// TIA Portal V17 program export: 1 tag tables, 0 data types, 3 data blocks, 7 code blocks (in call order from the OBs), 5 instance data blocks

VAR_GLOBAL   // PLC tag table "Default tag table"
   System_Byte AT %MB1 : Byte;
   FirstScan AT %M1.0 : Bool;
   DiagStatusUpdate AT %M1.1 : Bool;
   AlwaysTRUE AT %M1.2 : Bool;
   AlwaysFALSE AT %M1.3 : Bool;
   Clock_Byte AT %MB0 : Byte;
   Clock_10Hz AT %M0.0 : Bool;
   Clock_5Hz AT %M0.1 : Bool;
   "Clock_2.5Hz" AT %M0.2 : Bool;
   Clock_2Hz AT %M0.3 : Bool;
   "Clock_1.25Hz" AT %M0.4 : Bool;
   Clock_1Hz AT %M0.5 : Bool;
   "Clock_0.625Hz" AT %M0.6 : Bool;
   "Clock_0.5Hz" AT %M0.7 : Bool;
   lastEncoderValue AT %MW8 : Int;
   encoderNumberOfTurn AT %MD10 : DInt;
   machinePosition AT %MD14 : DInt;
   goToPosition AT %M2.0 : Bool;
   broken0 AT %Q0.0 : Bool;
   broken1 AT %Q0.1 : Bool;
   baseSensor AT %I0.0 : Bool;
   stepperMotor_Direction AT %Q0.3 : Bool;
   stepperMotor_Pulse AT %Q0.2 : Bool;
   jogBackward AT %M2.1 : Bool;
   baseReq AT %M2.2 : Bool;
   jogBackwardFromSetpoint AT %M2.3 : Bool;
   jogForward AT %M2.4 : Bool;
   jogForwardFromSetpoint AT %M2.5 : Bool;
   memoryBit0 AT %M2.6 : Bool;
   memoryBit1 AT %M2.7 : Bool;
   inPosition AT %M3.0 : Bool;
   memoryBit2 AT %M3.1 : Bool;
   memoryBit3 AT %M3.2 : Bool;
   homing AT %M3.3 : Bool;
   homingDone AT %M3.4 : Bool;
   memoryBit4 AT %M3.5 : Bool;
   memoryBit5 AT %M3.6 : Bool;
   homingStep1 AT %M3.7 : Bool;
   homingStep2 AT %M4.0 : Bool;
   memoryBit6 AT %M4.1 : Bool;
   homingStep3 AT %M4.2 : Bool;
   memoryBit7 AT %M4.3 : Bool;
   seqNum AT %MW6 : Int;
   memoryBit8 AT %M4.4 : Bool;
   memoryBit9 AT %M4.5 : Bool;
   memoryBit10 AT %M4.6 : Bool;
   checkPositionAfterReboot AT %M4.7 : Bool;
   memoryBit11 AT %M5.0 : Bool;
   positionNotActual AT %M5.1 : Bool;
END_VAR

DATA_BLOCK "HMI"   // DB2
{ S7_Optimized_Access := 'FALSE' }
VERSION : 0.1
// stored: AutoNumber true, DBAccessibleFromOPCUA true, IsOnlyStoredInLoadMemory false, IsWriteProtectedInAS false
   VAR RETAIN
      sensor : Bool := 1;
      machinePosition : DInt := 77;
      encoderTurn : DInt := 20;
      encoderPosition : Int;
      setpoint : Int;
      buttonBase : Bool;
      buttonStart : Bool;
      buttonStop : Bool;
      jogBackward : Bool;
      jogForward : Bool;
      jogVelocity : Int := 50;
      machineVelocity : Int := 70;
      baseVelocity : Int := 20;
      machineConst : DInt := 42625;   // numberOfpulseEncoder 1023 numberOfTurnPer90st 2,24*90
      serwisSetpointEnable : Bool;
      serwisMachineSetpoint : DInt;
   END_VAR
BEGIN
END_DATA_BLOCK

DATA_BLOCK "machineData"   // DB1
{ S7_Optimized_Access := 'TRUE' }
VERSION : 0.1
// stored: AutoNumber true, DBAccessibleFromOPCUA true, IsOnlyStoredInLoadMemory false, IsRetainMemResEnabled false, IsWriteProtectedInAS false, MemoryReserve 100
   VAR
      encoderTurn : DInt;
      reqVelocity : Real;
      encoderValue : Int;
   END_VAR
   VAR RETAIN
      machinePosition : DInt;
   END_VAR
   VAR
      direction : Bool;
   END_VAR
   VAR RETAIN
      lastEncoderValue : DInt;
      lastMachinePosition : DInt;
   END_VAR
BEGIN
END_DATA_BLOCK

DATA_BLOCK "modbus"   // DB3
{ S7_Optimized_Access := 'FALSE'; DB_Accessible_From_OPC_UA := 'FALSE' }
VERSION : 0.1
// stored: AutoNumber true, DBAccessibleFromOPCUA false, IsOnlyStoredInLoadMemory false, IsWriteProtectedInAS false
   VAR
      rs485parity : Int := 0;
      rs485baudrate : Int := 9600;
      modbusEncoderAdd : Int := 1;
      modbusMode : Int := 0;
      modbusEncoderDataRegister : DInt := 40001;
      modbusDataLength : DInt := 1;
      encoderMaxValue : DInt := 1024;
      mbLoadError : Bool;
      mbLoadDone : Bool;
      mbLoadStatus : Word;
      mbMasterBusy : Bool;
      mbMasterDone : Bool;
      mbMasterError : Bool;
      mbMasterStatus : Word;
      modbusReqBit : Bool;
      modbusReqAgainBit : Bool;
      modbusTimer : IEC_TIMER;
      REGISTERS : Array[0..9] of Int;
      lastEncoderValue : Int;
   END_VAR
BEGIN
   modbusTimer.PT := T#2S;
END_DATA_BLOCK

ORGANIZATION_BLOCK "Main"   // OB1, LAD, ProgramCycle
TITLE = "Main Program Sweep (Cycle)"
{ S7_Optimized_Access := 'TRUE' }
VERSION : 0.1
// stored: AutoNumber true, IsIECCheckEnabled false, SetENOAutomatically false
   VAR_INPUT
      Initial_Call : Bool;   // Initial call of this OB
      Remanence : Bool;   // =True, if remanent data are available
   END_VAR
   VAR_TEMP
      turn : Int;
      machinePosition : DInt;
   END_VAR
   VAR_TEMP   // added for the SCL form of the ladder/FBD networks
      _w1 : Bool;
      _w2 : Bool;
      _w3 : Bool;
   END_VAR
BEGIN

REGION Network 1: Encoder modbus function
   // te
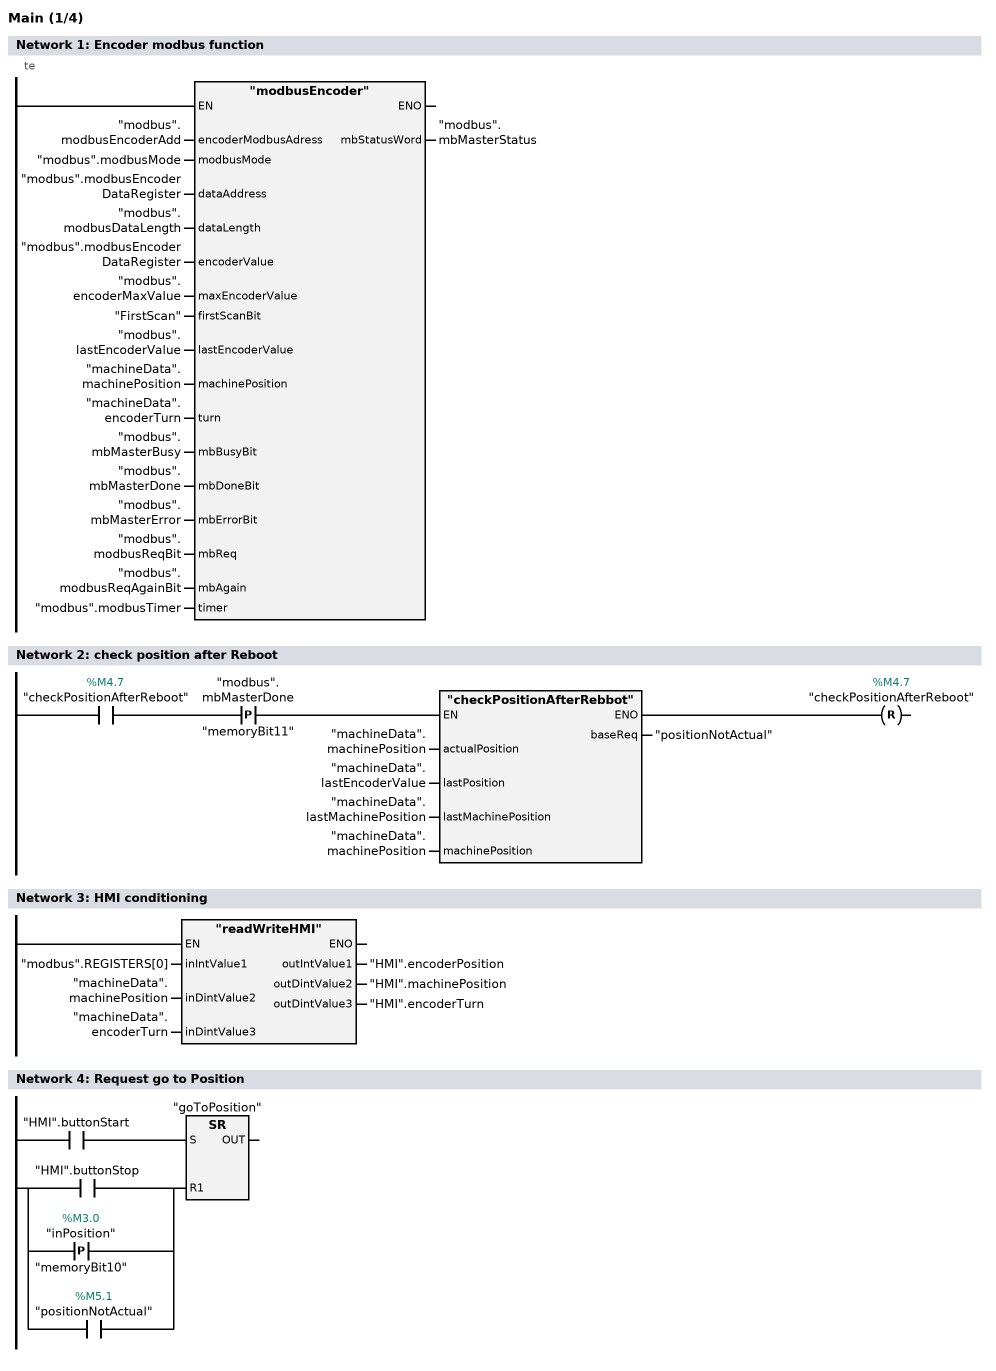
   RUNG wire#powerrail
      "modbusEncoder"(encoderModbusAdress := "modbus".modbusEncoderAdd, modbusMode := "modbus".modbusMode, dataAddress := "modbus".modbusEncoderDataRegister, dataLength := "modbus".modbusDataLength, encoderValue := "modbus".modbusEncoderDataRegister, maxEncoderValue := "modbus".encoderMaxValue, firstScanBit := "FirstScan", lastEncoderValue := "modbus".lastEncoderValue, machinePosition := "machineData".machinePosition, turn := "machineData".encoderTurn, mbBusyBit := "modbus".mbMasterBusy, mbDoneBit := "modbus".mbMasterDone, mbErrorBit := "modbus".mbMasterError, mbReq := "modbus".modbusReqBit, mbAgain := "modbus".modbusReqAgainBit, "timer" := "modbus".modbusTimer, mbStatusWord => "modbus".mbMasterStatus)
   END_RUNG
   // the same network as SCL:
   "modbusEncoder"(encoderModbusAdress := "modbus".modbusEncoderAdd,
                   modbusMode := "modbus".modbusMode,
                   dataAddress := "modbus".modbusEncoderDataRegister,
                   dataLength := "modbus".modbusDataLength,
                   encoderValue := "modbus".modbusEncoderDataRegister,
                   maxEncoderValue := "modbus".encoderMaxValue,
                   firstScanBit := "FirstScan",
                   lastEncoderValue := "modbus".lastEncoderValue,
                   machinePosition := "machineData".machinePosition,
                   turn := "machineData".encoderTurn,
                   mbBusyBit := "modbus".mbMasterBusy,
                   mbDoneBit := "modbus".mbMasterDone,
                   mbErrorBit := "modbus".mbMasterError,
                   mbReq := "modbus".modbusReqBit,
                   mbAgain := "modbus".modbusReqAgainBit,
                   "timer" := "modbus".modbusTimer,
                   mbStatusWord => "modbus".mbMasterStatus);
END_REGION

REGION Network 2: check position after Reboot
   RUNG wire#powerrail
      Contact( "checkPositionAfterReboot" )
      P_Contact(operand := "modbus".mbMasterDone, bit := "memoryBit11")
      "checkPositionAfterRebbot"(actualPosition := "machineData".machinePosition, lastPosition := "machineData".lastEncoderValue, lastMachinePosition := "machineData".lastMachinePosition, machinePosition := "machineData".machinePosition, baseReq => "positionNotActual")
      R_Coil( "checkPositionAfterReboot" )
   END_RUNG
   // the same network as SCL:
   #_w1 := "checkPositionAfterReboot" AND "modbus".mbMasterDone AND NOT "memoryBit11";   // rising edge of "modbus".mbMasterDone
   "memoryBit11" := "modbus".mbMasterDone;
   "checkPositionAfterRebbot"(EN := #_w1,
                           actualPosition := "machineData".machinePosition,
                           lastPosition := "machineData".lastEncoderValue,
                           lastMachinePosition := "machineData".lastMachinePosition,
                           machinePosition := "machineData".machinePosition,
                           baseReq => "positionNotActual",
                           ENO => #_w2);
   IF #_w2 THEN "checkPositionAfterReboot" := FALSE; END_IF;
END_REGION

REGION Network 3: HMI conditioning
   RUNG wire#powerrail
      "readWriteHMI"(inIntValue1 := "modbus".REGISTERS[0], inDintValue2 := "machineData".machinePosition, inDintValue3 := "machineData".encoderTurn, outIntValue1 => "HMI".encoderPosition, outDintValue2 => "HMI".machinePosition, outDintValue3 => "HMI".encoderTurn)
   END_RUNG
   // the same network as SCL:
   "readWriteHMI"(inIntValue1 := "modbus".REGISTERS[0],
                  inDintValue2 := "machineData".machinePosition,
                  inDintValue3 := "machineData".encoderTurn,
                  outIntValue1 => "HMI".encoderPosition,
                  outDintValue2 => "HMI".machinePosition,
                  outDintValue3 => "HMI".encoderTurn);
END_REGION

REGION Network 4: Request go to Position
   RUNG wire#powerrail
      Contact( "HMI".buttonStart )
      S_SR(operand := "goToPosition", r1 := wire#w1)
   END_RUNG
   RUNG wire#powerrail
      Contact( "HMI".buttonStop )
   END_RUNG wire#w1
   RUNG wire#powerrail
      P_Contact(operand := "inPosition", bit := "memoryBit10")
   END_RUNG wire#w1
   RUNG wire#powerrail
      Contact( "positionNotActual" )
   END_RUNG wire#w1
   // the same network as SCL:
   #_w1 := "inPosition" AND NOT "memoryBit10";   // rising edge of "inPosition"
   "memoryBit10" := "inPosition";
   IF "HMI".buttonStart THEN
       "goToPosition" := TRUE;   // SR flip-flop
   END_IF;
   IF "HMI".buttonStop OR #_w1 OR "positionNotActual" THEN "goToPosition" := FALSE; END_IF;
END_REGION

REGION Network 5: Homing
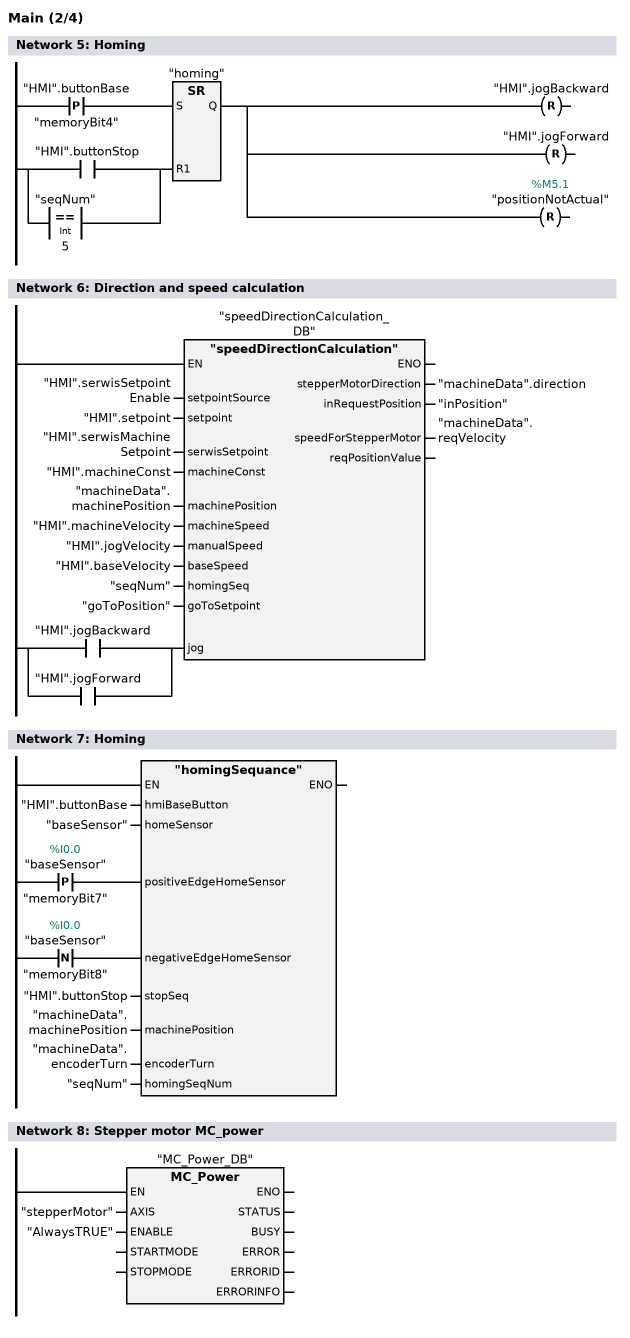
   RUNG wire#powerrail
      P_Contact(operand := "HMI".buttonBase, bit := "memoryBit4")
      S_SR(operand := "homing", r1 := wire#w1)
      wire#w2
      R_Coil( "HMI".jogBackward )
   END_RUNG
   RUNG wire#powerrail
      Contact( "HMI".buttonStop )
   END_RUNG wire#w1
   RUNG wire#powerrail
      { S7_Templates := "SrcType := Int" } EQ_Contact(in1 := "seqNum", in2 := 5)
   END_RUNG wire#w1
   RUNG wire#w2
      R_Coil( "HMI".jogForward )
   END_RUNG
   RUNG wire#w2
      R_Coil( "positionNotActual" )
   END_RUNG
   // the same network as SCL:
   #_w1 := "HMI".buttonBase AND NOT "memoryBit4";   // rising edge of "HMI".buttonBase
   "memoryBit4" := "HMI".buttonBase;
   IF #_w1 THEN
       "homing" := TRUE;   // SR flip-flop
   END_IF;
   IF "HMI".buttonStop OR ("seqNum" = 5) THEN "homing" := FALSE; END_IF;
   IF "homing" THEN
       "HMI".jogBackward := FALSE;
       "HMI".jogForward := FALSE;
       "positionNotActual" := FALSE;
   END_IF;
END_REGION

REGION Network 6: Direction and speed calculation
   RUNG wire#powerrail
      "speedDirectionCalculation_DB"(jog := wire#w1, setpointSource := "HMI".serwisSetpointEnable, setpoint := "HMI".setpoint, serwisSetpoint := "HMI".serwisMachineSetpoint, machineConst := "HMI".machineConst, machinePosition := "machineData".machinePosition, machineSpeed := "HMI".machineVelocity, manualSpeed := "HMI".jogVelocity, baseSpeed := "HMI".baseVelocity, homingSeq := "seqNum", goToSetpoint := "goToPosition", stepperMotorDirection => "machineData".direction, inRequestPosition => "inPosition", speedForStepperMotor => "machineData".reqVelocity, reqPositionValue =>)
   END_RUNG
   RUNG wire#powerrail
      Contact( "HMI".jogBackward )
   END_RUNG wire#w1
   RUNG wire#powerrail
      Contact( "HMI".jogForward )
   END_RUNG wire#w1
   // the same network as SCL:
   "speedDirectionCalculation_DB"(setpointSource := "HMI".serwisSetpointEnable,   // "speedDirectionCalculation"
                           setpoint := "HMI".setpoint,
                           serwisSetpoint := "HMI".serwisMachineSetpoint,
                           machineConst := "HMI".machineConst,
                           machinePosition := "machineData".machinePosition,
                           machineSpeed := "HMI".machineVelocity,
                           manualSpeed := "HMI".jogVelocity,
                           baseSpeed := "HMI".baseVelocity,
                           homingSeq := "seqNum",
                           goToSetpoint := "goToPosition",
                           jog := "HMI".jogBackward OR "HMI".jogForward,
                           stepperMotorDirection => "machineData".direction,
                           inRequestPosition => "inPosition",
                           speedForStepperMotor => "machineData".reqVelocity);
END_REGION

REGION Network 7: Homing
   RUNG wire#powerrail
      "homingSequance"(positiveEdgeHomeSensor := wire#w1, negativeEdgeHomeSensor := wire#w2, hmiBaseButton := "HMI".buttonBase, homeSensor := "baseSensor", stopSeq := "HMI".buttonStop, machinePosition := "machineData".machinePosition, encoderTurn := "machineData".encoderTurn, homingSeqNum := "seqNum")
   END_RUNG
   RUNG wire#powerrail
      P_Contact(operand := "baseSensor", bit := "memoryBit7")
   END_RUNG wire#w1
   RUNG wire#powerrail
      N_Contact(operand := "baseSensor", bit := "memoryBit8")
   END_RUNG wire#w2
   // the same network as SCL:
   #_w1 := "baseSensor" AND NOT "memoryBit7";   // rising edge of "baseSensor"
   "memoryBit7" := "baseSensor";
   #_w2 := NOT "baseSensor" AND "memoryBit8";   // falling edge of "baseSensor"
   "memoryBit8" := "baseSensor";
   "homingSequance"(hmiBaseButton := "HMI".buttonBase,
                    homeSensor := "baseSensor",
                    positiveEdgeHomeSensor := #_w1,
                    negativeEdgeHomeSensor := #_w2,
                    stopSeq := "HMI".buttonStop,
                    machinePosition := "machineData".machinePosition,
                    encoderTurn := "machineData".encoderTurn,
                    homingSeqNum := "seqNum");
END_REGION

REGION Network 8: Stepper motor MC_power
   RUNG wire#powerrail
      "MC_Power_DB".MC_Power(Axis := "stepperMotor", Enable := "AlwaysTRUE", StartMode :=, StopMode :=, Status =>, Busy =>, Error =>, ErrorID =>, ErrorInfo =>)
   END_RUNG
   // the same network as SCL:
   "MC_Power_DB"(Axis := "stepperMotor", Enable := "AlwaysTRUE");   // MC_Power
END_REGION

REGION Network 9: Srepper motor drive
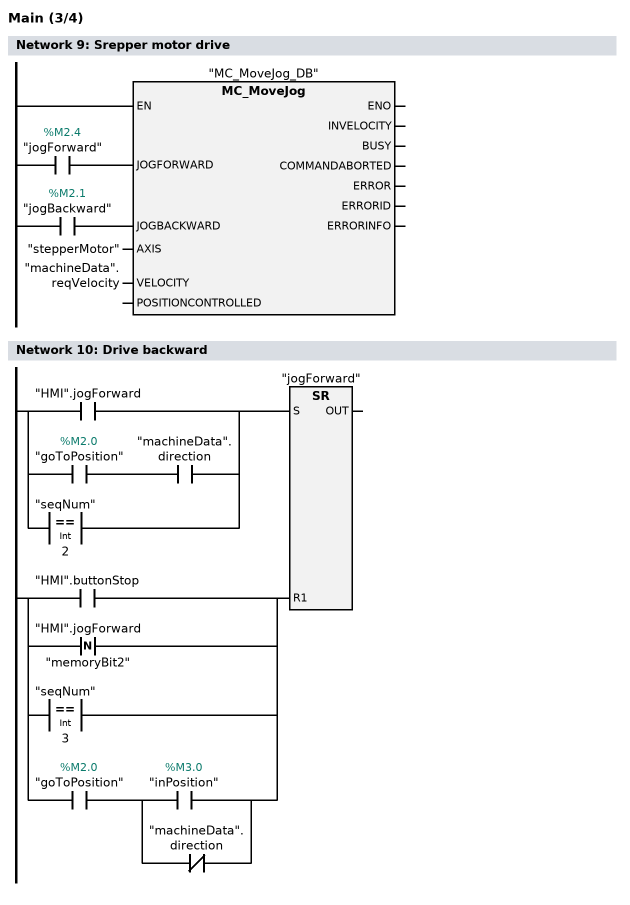
   RUNG wire#powerrail
      "MC_MoveJog_DB".MC_MoveJog(JogForward := wire#w1, JogBackward := wire#w2, Axis := "stepperMotor", Velocity := "machineData".reqVelocity, PositionControlled :=, InVelocity =>, Busy =>, CommandAborted =>, Error =>, ErrorID =>, ErrorInfo =>)
   END_RUNG
   RUNG wire#powerrail
      Contact( "jogForward" )
   END_RUNG wire#w1
   RUNG wire#powerrail
      Contact( "jogBackward" )
   END_RUNG wire#w2
   // the same network as SCL:
   "MC_MoveJog_DB"(JogForward := "jogForward",   // MC_MoveJog
                   JogBackward := "jogBackward",
                   Axis := "stepperMotor",
                   Velocity := "machineData".reqVelocity);
END_REGION

REGION Network 10: Drive backward
   RUNG wire#powerrail
      Contact( "HMI".jogForward )
      wire#w1
      S_SR(operand := "jogForward", r1 := wire#w3)
   END_RUNG
   RUNG wire#powerrail
      Contact( "goToPosition" )
      Contact( "machineData".direction )
   END_RUNG wire#w1
   RUNG wire#powerrail
      { S7_Templates := "SrcType := Int" } EQ_Contact(in1 := "seqNum", in2 := 2)
   END_RUNG wire#w1
   RUNG wire#powerrail
      Contact( "HMI".buttonStop )
   END_RUNG wire#w3
   RUNG wire#powerrail
      N_Contact(operand := "HMI".jogForward, bit := "memoryBit2")
   END_RUNG wire#w3
   RUNG wire#powerrail
      { S7_Templates := "SrcType := Int" } EQ_Contact(in1 := "seqNum", in2 := 3)
   END_RUNG wire#w3
   RUNG wire#powerrail
      Contact( "goToPosition" )
      wire#w2
      Contact( "inPosition" )
   END_RUNG wire#w3
   RUNG wire#w2
      I_Contact( "machineData".direction )
   END_RUNG wire#w3
   // the same network as SCL:
   #_w1 := NOT "HMI".jogForward AND "memoryBit2";   // falling edge of "HMI".jogForward
   "memoryBit2" := "HMI".jogForward;
   IF "HMI".jogForward OR ("goToPosition" AND "machineData".direction) OR ("seqNum" = 2) THEN
       "jogForward" := TRUE;   // SR flip-flop
   END_IF;
   IF "HMI".buttonStop OR #_w1 OR ("seqNum" = 3) OR ("goToPosition" AND ("inPosition" OR NOT "machineData".direction)) THEN
       "jogForward" := FALSE;
   END_IF;
END_REGION

REGION Network 11: Drive forward
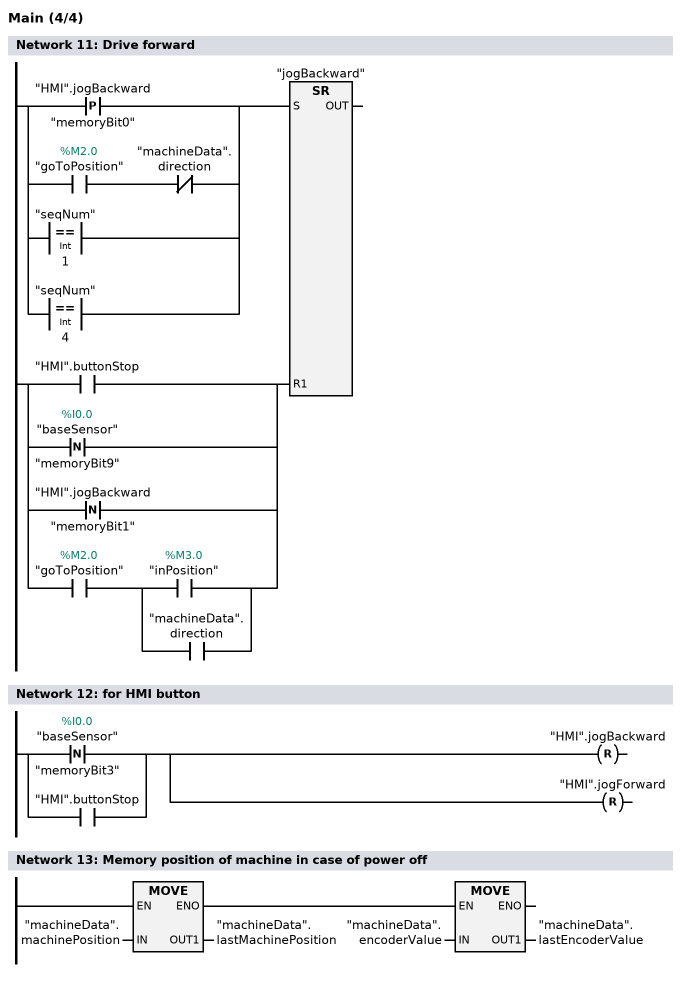
   RUNG wire#powerrail
      P_Contact(operand := "HMI".jogBackward, bit := "memoryBit0")
      wire#w1
      S_SR(operand := "jogBackward", r1 := wire#w3)
   END_RUNG
   RUNG wire#powerrail
      Contact( "goToPosition" )
      I_Contact( "machineData".direction )
   END_RUNG wire#w1
   RUNG wire#powerrail
      { S7_Templates := "SrcType := Int" } EQ_Contact(in1 := "seqNum", in2 := 1)
   END_RUNG wire#w1
   RUNG wire#powerrail
      { S7_Templates := "SrcType := Int" } EQ_Contact(in1 := "seqNum", in2 := 4)
   END_RUNG wire#w1
   RUNG wire#powerrail
      Contact( "HMI".buttonStop )
   END_RUNG wire#w3
   RUNG wire#powerrail
      N_Contact(operand := "baseSensor", bit := "memoryBit9")
   END_RUNG wire#w3
   RUNG wire#powerrail
      N_Contact(operand := "HMI".jogBackward, bit := "memoryBit1")
   END_RUNG wire#w3
   RUNG wire#powerrail
      Contact( "goToPosition" )
      wire#w2
      Contact( "inPosition" )
   END_RUNG wire#w3
   RUNG wire#w2
      Contact( "machineData".direction )
   END_RUNG wire#w3
   // the same network as SCL:
   #_w1 := "HMI".jogBackward AND NOT "memoryBit0";   // rising edge of "HMI".jogBackward
   "memoryBit0" := "HMI".jogBackward;
   #_w2 := NOT "baseSensor" AND "memoryBit9";   // falling edge of "baseSensor"
   "memoryBit9" := "baseSensor";
   #_w3 := NOT "HMI".jogBackward AND "memoryBit1";   // falling edge of "HMI".jogBackward
   "memoryBit1" := "HMI".jogBackward;
   IF #_w1 OR ("goToPosition" AND NOT "machineData".direction) OR ("seqNum" = 1) OR ("seqNum" = 4) THEN
       "jogBackward" := TRUE;   // SR flip-flop
   END_IF;
   IF "HMI".buttonStop OR #_w2 OR #_w3 OR ("goToPosition" AND ("inPosition" OR "machineData".direction)) THEN
       "jogBackward" := FALSE;
   END_IF;
END_REGION

REGION Network 12: for HMI button
   RUNG wire#powerrail
      N_Contact(operand := "baseSensor", bit := "memoryBit3")
      wire#w1
      R_Coil( "HMI".jogBackward )
   END_RUNG
   RUNG wire#powerrail
      Contact( "HMI".buttonStop )
   END_RUNG wire#w1
   RUNG wire#w1
      R_Coil( "HMI".jogForward )
   END_RUNG
   // the same network as SCL:
   #_w1 := NOT "baseSensor" AND "memoryBit3";   // falling edge of "baseSensor"
   "memoryBit3" := "baseSensor";
   IF #_w1 OR "HMI".buttonStop THEN
       "HMI".jogBackward := FALSE;
       "HMI".jogForward := FALSE;
   END_IF;
END_REGION

REGION Network 13: Memory position of machine in case of power off
   RUNG wire#powerrail
      Move(in := "machineData".machinePosition, out1 => "machineData".lastMachinePosition)
      Move(in := "machineData".encoderValue, out1 => "machineData".lastEncoderValue)
   END_RUNG
   // the same network as SCL:
   "machineData".lastMachinePosition := "machineData".machinePosition;
   "machineData".lastEncoderValue := "machineData".encoderValue;
END_REGION
END_ORGANIZATION_BLOCK

FUNCTION "modbusEncoder" : Void   // FC1, LAD
{ S7_Optimized_Access := 'TRUE' }
VERSION : 0.1
// stored: AutoNumber true, IsIECCheckEnabled false, SetENOAutomatically false, UDAEnableTagReadback false
   VAR_INPUT
      encoderModbusAdress : UInt;
      modbusMode : USInt;   // modbus mode; 0- read holding register(03);1-Writing a holding register; see help MB_Master
      dataAddress : UDInt;   // starting adress (40001)
      dataLength : UDInt;
      encoderValue : Int;
      maxEncoderValue : Int;
      firstScanBit : Bool;
   END_VAR
   VAR_OUTPUT
      mbStatusWord : Word;
   END_VAR
   VAR_IN_OUT
      lastEncoderValue : Int;
      machinePosition : DInt;
      turn : DInt;
      mbBusyBit : Bool;
      mbDoneBit : Bool;
      mbErrorBit : Bool;
      mbReq : Bool;
      mbAgain : Bool;
      "timer" : IEC_TIMER;
   END_VAR
   VAR_TEMP
      rotationDistance : DInt;
   END_VAR
BEGIN

REGION Network 1: Modbus data block
   // Pobranie danych po modbusie do bloku danych
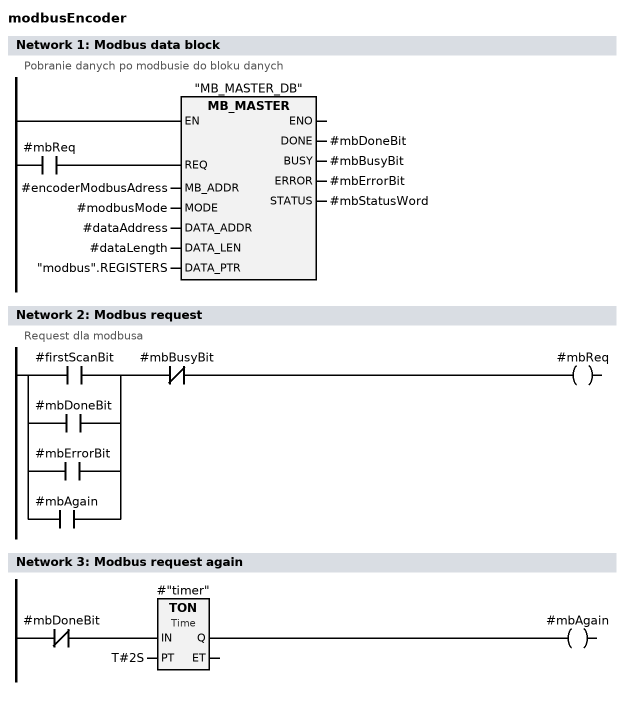
   RUNG wire#powerrail
      "MB_MASTER_DB".MB_MASTER(REQ := wire#w1, MB_ADDR := #encoderModbusAdress, MODE := #modbusMode, DATA_ADDR := #dataAddress, DATA_LEN := #dataLength, DATA_PTR := "modbus".REGISTERS, DONE => #mbDoneBit, BUSY => #mbBusyBit, ERROR => #mbErrorBit, STATUS => #mbStatusWord)
   END_RUNG
   RUNG wire#powerrail
      Contact( #mbReq )
   END_RUNG wire#w1
   // the same network as SCL:
   "MB_MASTER_DB"(REQ := #mbReq,   // MB_MASTER
                  MB_ADDR := #encoderModbusAdress,
                  MODE := #modbusMode,
                  DATA_ADDR := #dataAddress,
                  DATA_LEN := #dataLength,
                  DATA_PTR := "modbus".REGISTERS,
                  DONE => #mbDoneBit,
                  BUSY => #mbBusyBit,
                  ERROR => #mbErrorBit,
                  STATUS => #mbStatusWord);
END_REGION

REGION Network 2: Modbus request
   // Request dla modbusa
   RUNG wire#powerrail
      Contact( #firstScanBit )
      wire#w1
      I_Contact( #mbBusyBit )
      Coil( #mbReq )
   END_RUNG
   RUNG wire#powerrail
      Contact( #mbDoneBit )
   END_RUNG wire#w1
   RUNG wire#powerrail
      Contact( #mbErrorBit )
   END_RUNG wire#w1
   RUNG wire#powerrail
      Contact( #mbAgain )
   END_RUNG wire#w1
   // the same network as SCL:
   #mbReq := (#firstScanBit OR #mbDoneBit OR #mbErrorBit OR #mbAgain) AND NOT #mbBusyBit;
END_REGION

REGION Network 3: Modbus request again
   RUNG wire#powerrail
      I_Contact( #mbDoneBit )
      { S7_Templates := "time_type := Time" } #"timer".TON(pt := T#2S, et =>)
      Coil( #mbAgain )
   END_RUNG
   // the same network as SCL:
   #"timer".TON(IN := NOT #mbDoneBit, PT := T#2S);
   #mbAgain := #"timer".Q;
END_REGION

REGION Network 4 (SCL)
   #encoderValue := "modbus".REGISTERS[0];
   IF (#encoderValue <> #lastEncoderValue) THEN
       #rotationDistance := #encoderValue - #lastEncoderValue;
       IF (#rotationDistance > (#maxEncoderValue / 2)) THEN
           #turn := #turn - 1;
       ELSIF (#rotationDistance < ((-1) * #maxEncoderValue / 2)) THEN
           #turn := #turn + 1;
       END_IF;

       #machinePosition := #turn * #maxEncoderValue + #encoderValue;
       #lastEncoderValue := #encoderValue;

   END_IF;
END_REGION
END_FUNCTION

FUNCTION "checkPositionAfterRebbot" : Void
{ S7_Optimized_Access := 'TRUE' }
VERSION : 0.1
   VAR_INPUT 
      actualPosition : DInt;
      lastPosition : DInt;
      lastMachinePosition : DInt;
   END_VAR

   VAR_OUTPUT 
      baseReq : Bool;
   END_VAR

   VAR_IN_OUT 
      machinePosition : DInt;
   END_VAR

   VAR_TEMP 
      lowPositionLimit : DInt;
      highPositionLimit : DInt;
   END_VAR


BEGIN
	    #lowPositionLimit := #lastPosition - 1;
	    #highPositionLimit := #lastPosition + 1;
	    IF (#actualPosition>=#lowPositionLimit & #actualPosition<#highPositionLimit) THEN
	        #baseReq := 0;
	        #machinePosition := #lastMachinePosition;
	    ELSE
	        #baseReq := 1;
	        ;
	    END_IF;
	    
	
	
END_FUNCTION

FUNCTION "readWriteHMI" : Void
{ S7_Optimized_Access := 'TRUE' }
VERSION : 0.1
   VAR_INPUT 
      inIntValue1 : Int;
      inDintValue2 : DInt;
      inDintValue3 : DInt;
   END_VAR

   VAR_OUTPUT 
      outIntValue1 : Int;
      outDintValue2 : DInt;
      outDintValue3 : DInt;
   END_VAR


BEGIN
	#outIntValue1 := #inIntValue1;
	#outDintValue2 := #inDintValue2;
	#outDintValue3 := #inDintValue3;
	
END_FUNCTION

FUNCTION_BLOCK "speedDirectionCalculation"
{ S7_Optimized_Access := 'TRUE' }
VERSION : 0.1
   VAR_INPUT 
      setpointSource : Bool;   // set in HMI, 0-user setpoint in st, 1-serwis setpoint in machine position value
      setpoint : Int;   // setpoint in st
      serwisSetpoint : DInt;
      machineConst : Real;
      machinePosition : DInt;
      machineSpeed : Int;
      manualSpeed : Int;
      baseSpeed : Int;
      homingSeq : Int;
      goToSetpoint : Bool;
      jog : Bool;
   END_VAR

   VAR_OUTPUT 
      stepperMotorDirection : Bool;
      inRequestPosition : Bool;
      speedForStepperMotor : Real;
      reqPositionValue : DInt := 0;
   END_VAR

   VAR 
      reqPosition : Real;
   END_VAR

   VAR_TEMP 
      diff : DInt;
      distanceToDrive : DInt;
   END_VAR


BEGIN
	#reqPositionValue := 0;
	IF #setpointSource = TRUE THEN
	    #reqPositionValue := #serwisSetpoint;
	ELSE
	    #reqPosition := (INT_TO_REAL(#setpoint) + 450.0) / 900.0 * #machineConst;
	    #reqPositionValue := REAL_TO_DINT(#reqPosition);
	END_IF;
	
	#inRequestPosition := false;
	
	IF #reqPositionValue<#machinePosition THEN
	    #stepperMotorDirection := false;
	   // Statement section IF
	ELSIF (#reqPositionValue>#machinePosition) THEN
	    #stepperMotorDirection := true;
	ELSE
	    #inRequestPosition := true;
	END_IF;
	
	//speed calculation
	//
	IF (#goToSetpoint = 1) THEN
	    #speedForStepperMotor := INT_TO_REAL(#machineSpeed) / 50;
	    #diff := ABS(#reqPositionValue - #machinePosition);
	    
	    IF (#diff < 100) THEN
	        #speedForStepperMotor := INT_TO_REAL(#machineSpeed) / 400;
	        IF (#diff < 10) THEN
	            #speedForStepperMotor := INT_TO_REAL(#machineSpeed) / 1200;
	        END_IF;
	    END_IF;
	ELSIF #jog = 1 THEN
	    #speedForStepperMotor := INT_TO_REAL(#manualSpeed) / 100;
	ELSIF #homingSeq = 1 THEN
	    #speedForStepperMotor := INT_TO_REAL(#baseSpeed) / 100; //predkość szybka powrotu
	ELSIF #homingSeq =2 THEN
	    #speedForStepperMotor := INT_TO_REAL(#baseSpeed) / 200; //predkość odjazdu
	ELSIF #homingSeq =4 THEN
	    #speedForStepperMotor := INT_TO_REAL(#baseSpeed) / 800;
	    
	ELSE
	    #speedForStepperMotor := 0.1;
	END_IF;
	    
	    
	    
	    
	
END_FUNCTION_BLOCK

FUNCTION "homingSequance" : Void
{ S7_Optimized_Access := 'TRUE' }
VERSION : 0.1
   VAR_INPUT 
      hmiBaseButton : Bool;
      homeSensor : Bool;
      positiveEdgeHomeSensor : Bool;
      negativeEdgeHomeSensor : Bool;
      stopSeq : Bool;
   END_VAR

   VAR_IN_OUT 
      machinePosition : DInt;
      encoderTurn : DInt;
      homingSeqNum : Int;
   END_VAR


BEGIN
	IF (#hmiBaseButton = TRUE & #homingSeqNum=0 & #homeSensor=true) THEN
	    #homingSeqNum := 1; //start bazowania
	ELSIF (#homingSeqNum = 1 & #negativeEdgeHomeSensor = TRUE) THEN
	    #homingSeqNum := 2; //wykrycie czujnika home i zatrzymanie
	ELSIF (#homingSeqNum = 2 & #positiveEdgeHomeSensor = TRUE) THEN
	    #homingSeqNum := 3; // zjazd z czujnika
	ELSIF (#homingSeqNum = 3) THEN
	    #homingSeqNum := 4;//ponowny dojazd
	ELSIF (#homingSeqNum = 4 & #negativeEdgeHomeSensor = TRUE) THEN
	    #homingSeqNum := 5;//zatrzymanie
	    
	ELSIF #homingSeqNum = 5 THEN
	    #homingSeqNum := 0;
	   // #machinePosition := 0;
	  //  #encoderTurn := 0; //na czas testów wykomentowano
	END_IF;
	IF (#stopSeq = true) THEN
	    #homingSeqNum := 0;
	END_IF;
	
	    
	
END_FUNCTION

ORGANIZATION_BLOCK "Startup"   // OB100, LAD, Startup
TITLE = "Complete Restart"
{ S7_Optimized_Access := 'TRUE' }
VERSION : 0.1
// stored: AutoNumber true, IsIECCheckEnabled false, SetENOAutomatically false
   VAR_INPUT
      LostRetentive : Bool;   // True if retentive data are lost
      LostRTC : Bool;   // True if date and time are lost
   END_VAR
BEGIN

REGION Network 1: modbus Master Init
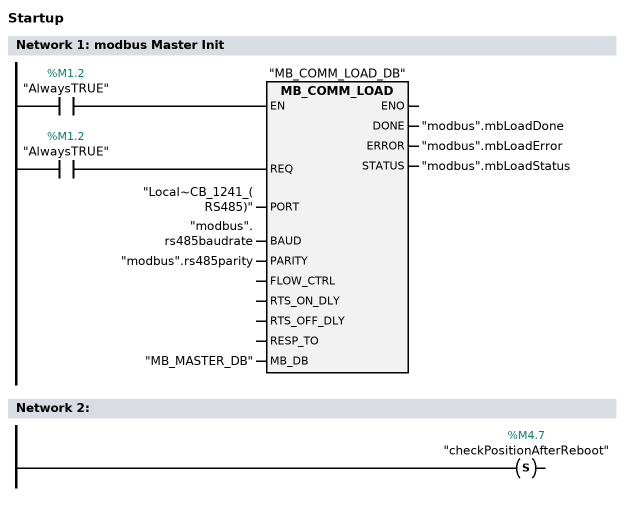
   RUNG wire#powerrail
      Contact( "AlwaysTRUE" )
      "MB_COMM_LOAD_DB".MB_COMM_LOAD(REQ := wire#w1, PORT := "Local~CB_1241_(RS485)", BAUD := "modbus".rs485baudrate, PARITY := "modbus".rs485parity, FLOW_CTRL :=, RTS_ON_DLY :=, RTS_OFF_DLY :=, RESP_TO :=, MB_DB := "MB_MASTER_DB", DONE => "modbus".mbLoadDone, ERROR => "modbus".mbLoadError, STATUS => "modbus".mbLoadStatus)
   END_RUNG
   RUNG wire#powerrail
      Contact( "AlwaysTRUE" )
   END_RUNG wire#w1
   // the same network as SCL:
   IF "AlwaysTRUE" THEN
       "MB_COMM_LOAD_DB"(REQ := "AlwaysTRUE",   // MB_COMM_LOAD
                         PORT := "Local~CB_1241_(RS485)",
                         BAUD := "modbus".rs485baudrate,
                         PARITY := "modbus".rs485parity,
                         MB_DB := "MB_MASTER_DB",
                         DONE => "modbus".mbLoadDone,
                         ERROR => "modbus".mbLoadError,
                         STATUS => "modbus".mbLoadStatus);
   END_IF;
END_REGION

REGION Network 2
   RUNG wire#powerrail
      S_Coil( "checkPositionAfterReboot" )
   END_RUNG
   // the same network as SCL:
   "checkPositionAfterReboot" := TRUE;
END_REGION
END_ORGANIZATION_BLOCK

DATA_BLOCK "speedDirectionCalculation_DB"   // DB9
VERSION : 0.1
// stored: AutoNumber true, DBAccessibleFromOPCUA true, InstanceOfName speedDirectionCalculation, InstanceOfType FB
"speedDirectionCalculation"
BEGIN
END_DATA_BLOCK

DATA_BLOCK "MB_COMM_LOAD_DB"   // DB4
// stored: AutoNumber true, DBAccessibleFromOPCUA true, InstanceOfName MB_COMM_LOAD, OfSystemLibElement MB_COMM_LOAD, OfSystemLibVersion 2.1
"MB_COMM_LOAD"
   // VAR_INPUT
   //    REQ : Bool;
   //    PORT : PORT;
   //    BAUD : UDInt;
   //    PARITY : UInt;
   //    FLOW_CTRL : UInt;
   //    RTS_ON_DLY : UInt;
   //    RTS_OFF_DLY : UInt;
   //    RESP_TO : UInt;
   // END_VAR
   // VAR_OUTPUT
   //    DONE : Bool;
   //    ERROR : Bool;
   //    STATUS : Word;
   // END_VAR
   // VAR_IN_OUT
   //    MB_DB : MB_BASE;
   // END_VAR
   // VAR
   //    ICHAR_GAP : UInt;
   //    RETRIES : UInt;
   //    WRREC_STATUS : Word;
   //    RDREC_STATUS : Word;
   //    SFC_STATUS : Word;
   //    Port_CFG_SFB : Array[0..25] of Byte;
   //    Send_CFG_SFB : Array[0..16] of Byte;
   //    Rcv_CFG_SFB : Array[0..60] of Byte;
   //    STOP_BITS : USInt;
   // END_VAR
BEGIN
END_DATA_BLOCK

DATA_BLOCK "MB_MASTER_DB"   // DB5
// stored: AutoNumber true, DBAccessibleFromOPCUA true, InstanceOfName MB_MASTER, OfSystemLibElement MB_MASTER, OfSystemLibVersion 2.2
"MB_MASTER"
   // // inherited from MB_BASE
   // VAR
   //    S_PORT : UInt;
   //    S_RESP_TO : UInt;
   //    S_ICHAR_GAP : UInt;
   //    S_RETRIES : UInt;
   // END_VAR
   // VAR_INPUT
   //    REQ : Bool;
   //    MB_ADDR : UInt;
   //    MODE : USInt;
   //    DATA_ADDR : UDInt;
   //    DATA_LEN : UInt;
   // END_VAR
   // VAR_OUTPUT
   //    DONE : Bool;
   //    BUSY : Bool;
   //    ERROR : Bool;
   //    STATUS : Word;
   // END_VAR
   // VAR_IN_OUT
   //    DATA_PTR : Variant;
   // END_VAR
   // VAR
   //    SEND_PTP_SFB : Array[0..11] of Byte;
   //    RCV_PTP_SFB : Array[0..11] of Byte;
   //    RCV_RST_SFB : Array[0..9] of Byte;
   //    PF_FREQUENCY : Real;
   //    BLOCKED_PROC_TIMEOUT : Real;
   //    CURRENT_TIME_VALUE : UDInt;
   //    SAVED_TIME_VALUE : UDInt;
   //    SAVED_SLAVE_ADDR : Word;
   //    SAVED_MODE : Word;
   //    SAVED_DATA_ADDR : DWord;
   //    SAVED_DATA_LEN : UInt;
   //    MB_STATE : UInt;
   //    COMM_SENT_COUNT : UInt;
   //    BYTE_COUNT : USInt;
   //    INIT_OK : Bool;
   //    ACTIVE : Bool;
   //    BROADCAST_FLAG : Bool;
   //    EXTENDED_ADDRESSING : Bool;
   //    SAVED_START_ADDR : UInt;
   //    TXBuf_Function_Offset : UDInt;
   //    TXBuf_Address_Offset : UDInt;
   //    TXBuf_Quantity_Offset : UDInt;
   // END_VAR
BEGIN
END_DATA_BLOCK

DATA_BLOCK "MC_MoveJog_DB"   // DB8
// stored: AutoNumber true, DBAccessibleFromOPCUA true, InstanceOfName MC_MoveJog, OfSystemLibElement MC_MoveJog, OfSystemLibVersion 8.0
"MC_MoveJog"
   // VAR_INPUT
   //    Axis : TO_SpeedAxis;
   //    JogForward : Bool;
   //    JogBackward : Bool;
   //    Velocity : Real;
   //    PositionControlled : Bool;
   // END_VAR
   // VAR_OUTPUT
   //    InVelocity : Bool;
   //    Busy : Bool;
   //    CommandAborted : Bool;
   //    Error : Bool;
   //    ErrorID : Word;
   //    ErrorInfo : Word;
   // END_VAR
   // VAR
   //    FB_ID : DInt;
   // END_VAR
BEGIN
END_DATA_BLOCK

DATA_BLOCK "MC_Power_DB"   // DB7
// stored: AutoNumber true, DBAccessibleFromOPCUA true, InstanceOfName MC_Power, OfSystemLibElement MC_Power, OfSystemLibVersion 8.0
"MC_Power"
   // VAR_INPUT
   //    Axis : TO_Axis;
   //    Enable : Bool;
   //    StartMode : Int;
   //    StopMode : Int;
   // END_VAR
   // VAR_OUTPUT
   //    Status : Bool;
   //    Busy : Bool;
   //    Error : Bool;
   //    ErrorID : Word;
   //    ErrorInfo : Word;
   // END_VAR
   // VAR
   //    FB_ID : DInt;
   // END_VAR
BEGIN
END_DATA_BLOCK
